% RSLogix 500 project I2P JOB 15 - SOLUTION.RSS, saved by version 10.00.00.00 %
PROJECT "UNTITLED"    % processor: Bul.1763 MicroLogix 1100 Series B %

PROGRAM FILES
  LAD 2   16 rungs

DATA FILES
  O0 OUTPUT  4 elements
  I1 INPUT  6 elements
  S2 STATUS  66 elements
  B3 BINARY  1 elements
  T4 TIMER  1 elements
  C5 COUNTER  1 elements
  R6 CONTROL  1 elements
  N7 INTEGER  1 elements
  F8 FLOAT  1 elements

LADDER 2
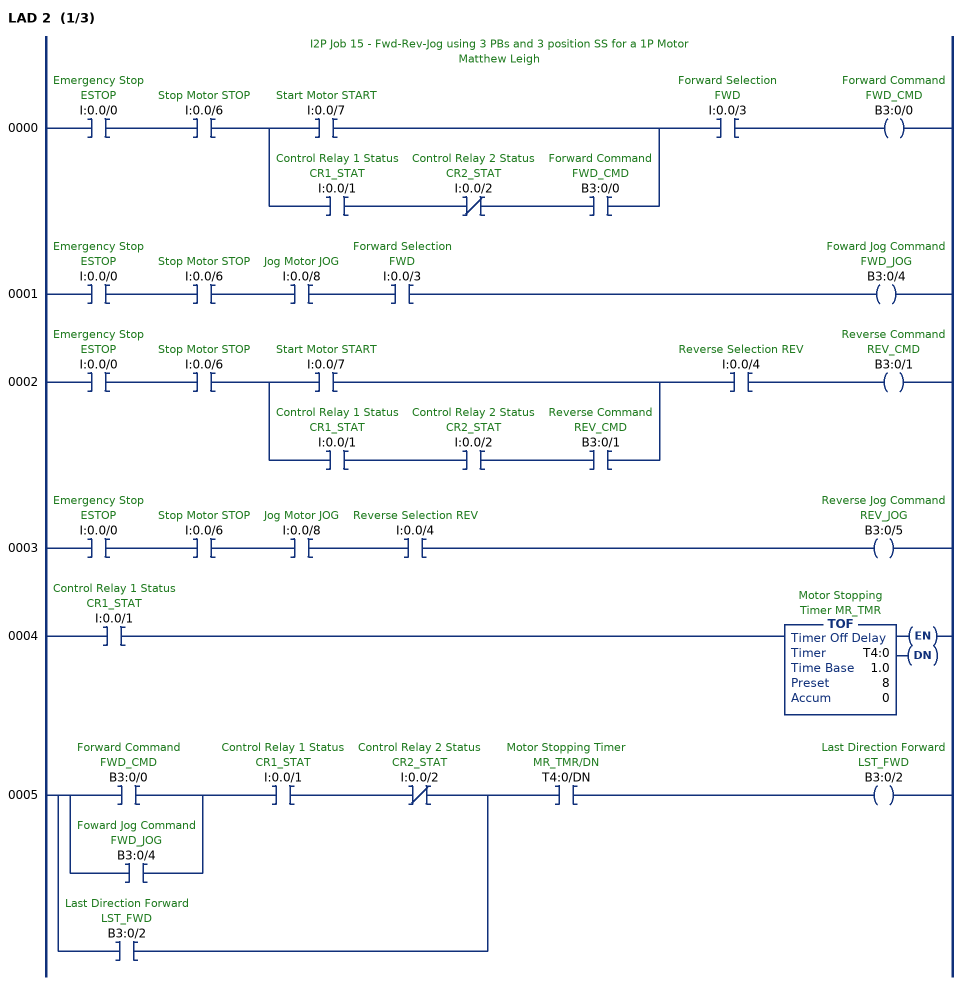
% Rung: 0 %
% I2P Job 15 - Fwd-Rev-Jog using 3 PBs and 3 position SS for a 1P Motor
% Matthew Leigh %
SOR XIC I:0.0/0 XIC I:0.0/6 BST XIC I:0.0/7 NXB XIC I:0.0/1 XIO I:0.0/2 XIC B3:0/0 BND XIC I:0.0/3 OTE B3:0/0 EOR
%   I:0.0/0  ESTOP  "Emergency Stop" %
%   I:0.0/6  STOP  "Stop Motor" %
%   I:0.0/7  START  "Start Motor" %
%   I:0.0/1  CR1_STAT  "Control Relay 1 Status" %
%   I:0.0/2  CR2_STAT  "Control Relay 2 Status" %
%   B3:0/0  FWD_CMD  "Forward Command" %
%   I:0.0/3  FWD  "Forward Selection" %
% Rung: 1 %
SOR XIC I:0.0/0 XIC I:0.0/6 XIC I:0.0/8 XIC I:0.0/3 OTE B3:0/4 EOR
%   I:0.0/0  ESTOP  "Emergency Stop" %
%   I:0.0/6  STOP  "Stop Motor" %
%   I:0.0/8  JOG  "Jog Motor" %
%   I:0.0/3  FWD  "Forward Selection" %
%   B3:0/4  FWD_JOG  "Foward Jog Command" %
% Rung: 2 %
SOR XIC I:0.0/0 XIC I:0.0/6 BST XIC I:0.0/7 NXB XIC I:0.0/1 XIC I:0.0/2 XIC B3:0/1 BND XIC I:0.0/4 OTE B3:0/1 EOR
%   I:0.0/0  ESTOP  "Emergency Stop" %
%   I:0.0/6  STOP  "Stop Motor" %
%   I:0.0/7  START  "Start Motor" %
%   I:0.0/1  CR1_STAT  "Control Relay 1 Status" %
%   I:0.0/2  CR2_STAT  "Control Relay 2 Status" %
%   B3:0/1  REV_CMD  "Reverse Command" %
%   I:0.0/4  REV  "Reverse Selection" %
% Rung: 3 %
SOR XIC I:0.0/0 XIC I:0.0/6 XIC I:0.0/8 XIC I:0.0/4 OTE B3:0/5 EOR
%   I:0.0/0  ESTOP  "Emergency Stop" %
%   I:0.0/6  STOP  "Stop Motor" %
%   I:0.0/8  JOG  "Jog Motor" %
%   I:0.0/4  REV  "Reverse Selection" %
%   B3:0/5  REV_JOG  "Reverse Jog Command" %
% Rung: 4 %
SOR XIC I:0.0/1 TOF T4:0 1.0 8 0 EOR
%   I:0.0/1  CR1_STAT  "Control Relay 1 Status" %
%   T4:0  MR_TMR  "Motor Stopping Timer" %
% Rung: 5 %
SOR BST BST XIC B3:0/0 NXB XIC B3:0/4 BND XIC I:0.0/1 XIO I:0.0/2 NXB XIC B3:0/2 BND XIC T4:0/DN OTE B3:0/2 EOR
%   B3:0/0  FWD_CMD  "Forward Command" %
%   B3:0/4  FWD_JOG  "Foward Jog Command" %
%   I:0.0/1  CR1_STAT  "Control Relay 1 Status" %
%   I:0.0/2  CR2_STAT  "Control Relay 2 Status" %
%   B3:0/2  LST_FWD  "Last Direction Forward" %
%   T4:0  MR_TMR  "Motor Stopping Timer" %

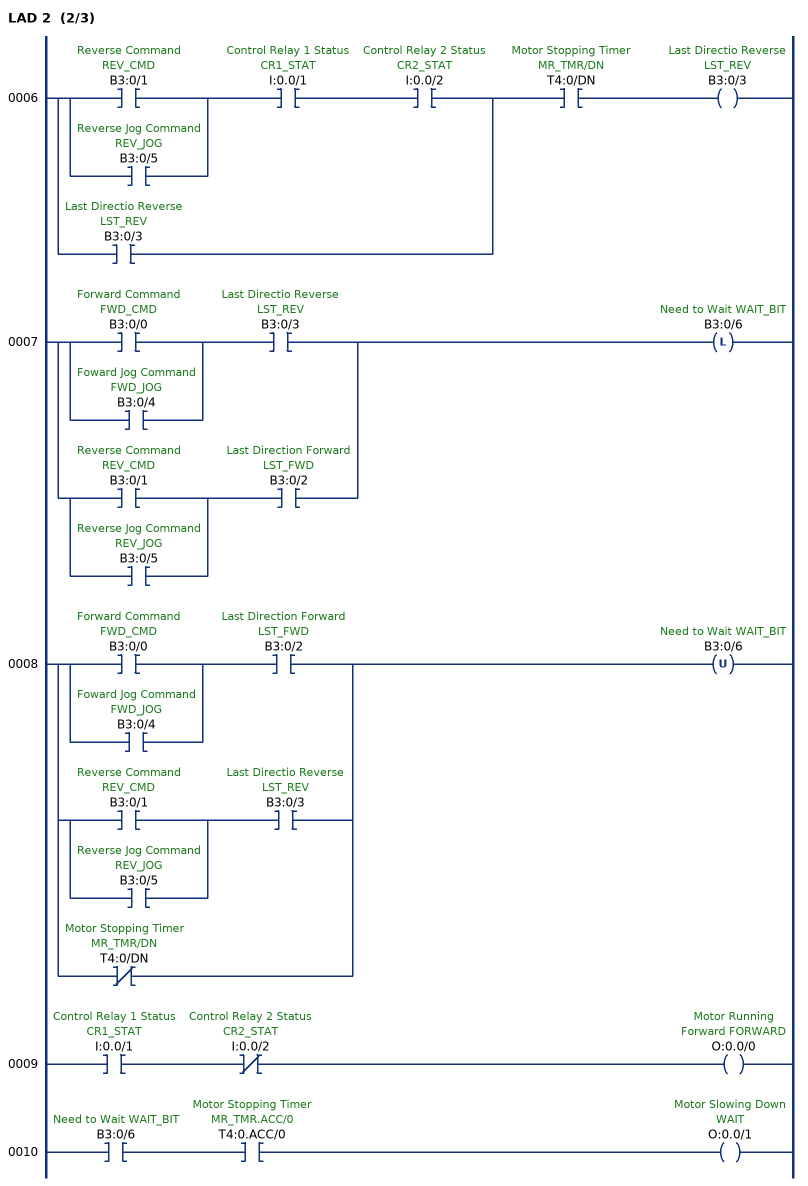
% Rung: 6 %
SOR BST BST XIC B3:0/1 NXB XIC B3:0/5 BND XIC I:0.0/1 XIC I:0.0/2 NXB XIC B3:0/3 BND XIC T4:0/DN OTE B3:0/3 EOR
%   B3:0/1  REV_CMD  "Reverse Command" %
%   B3:0/5  REV_JOG  "Reverse Jog Command" %
%   I:0.0/1  CR1_STAT  "Control Relay 1 Status" %
%   I:0.0/2  CR2_STAT  "Control Relay 2 Status" %
%   B3:0/3  LST_REV  "Last Directio Reverse" %
%   T4:0  MR_TMR  "Motor Stopping Timer" %
% Rung: 7 %
SOR BST BST XIC B3:0/0 NXB XIC B3:0/4 BND XIC B3:0/3 NXB BST XIC B3:0/1 NXB XIC B3:0/5 BND XIC B3:0/2 BND OTL B3:0/6 EOR
%   B3:0/0  FWD_CMD  "Forward Command" %
%   B3:0/4  FWD_JOG  "Foward Jog Command" %
%   B3:0/3  LST_REV  "Last Directio Reverse" %
%   B3:0/1  REV_CMD  "Reverse Command" %
%   B3:0/5  REV_JOG  "Reverse Jog Command" %
%   B3:0/2  LST_FWD  "Last Direction Forward" %
%   B3:0/6  WAIT_BIT  "Need to Wait" %
% Rung: 8 %
SOR BST BST XIC B3:0/0 NXB XIC B3:0/4 BND XIC B3:0/2 NXB BST XIC B3:0/1 NXB XIC B3:0/5 BND XIC B3:0/3 NXB XIO T4:0/DN BND OTU B3:0/6 EOR
%   B3:0/0  FWD_CMD  "Forward Command" %
%   B3:0/4  FWD_JOG  "Foward Jog Command" %
%   B3:0/2  LST_FWD  "Last Direction Forward" %
%   B3:0/1  REV_CMD  "Reverse Command" %
%   B3:0/5  REV_JOG  "Reverse Jog Command" %
%   B3:0/3  LST_REV  "Last Directio Reverse" %
%   T4:0  MR_TMR  "Motor Stopping Timer" %
%   B3:0/6  WAIT_BIT  "Need to Wait" %
% Rung: 9 %
SOR XIC I:0.0/1 XIO I:0.0/2 OTE O:0.0/0 EOR
%   I:0.0/1  CR1_STAT  "Control Relay 1 Status" %
%   I:0.0/2  CR2_STAT  "Control Relay 2 Status" %
%   O:0.0/0  FORWARD  "Motor Running Forward" %
% Rung: 10 %
SOR XIC B3:0/6 XIC T4:0.ACC/0 OTE O:0.0/1 EOR
%   B3:0/6  WAIT_BIT  "Need to Wait" %
%   T4:0  MR_TMR  "Motor Stopping Timer" %
%   O:0.0/1  WAIT  "Motor Slowing Down" %

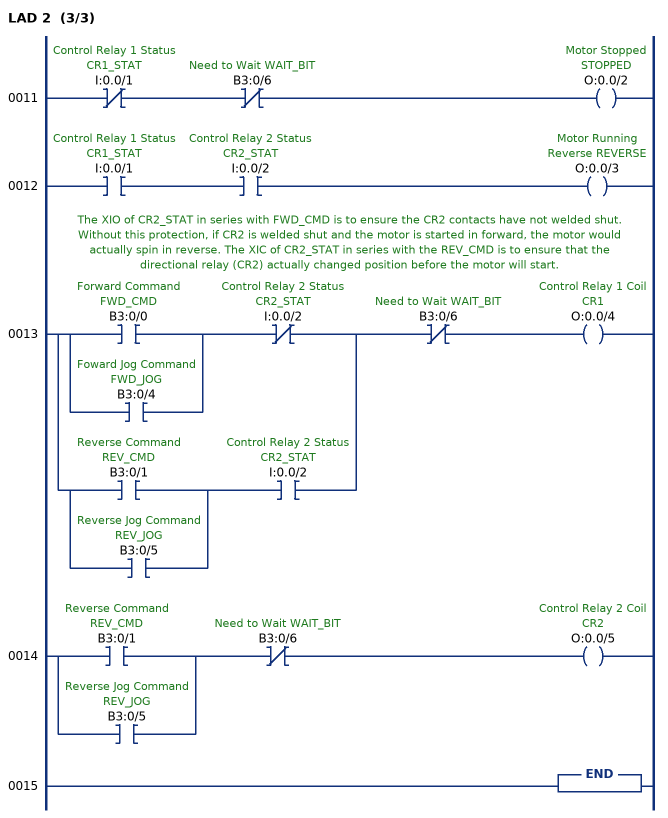
% Rung: 11 %
SOR XIO I:0.0/1 XIO B3:0/6 OTE O:0.0/2 EOR
%   I:0.0/1  CR1_STAT  "Control Relay 1 Status" %
%   B3:0/6  WAIT_BIT  "Need to Wait" %
%   O:0.0/2  STOPPED  "Motor Stopped" %
% Rung: 12 %
SOR XIC I:0.0/1 XIC I:0.0/2 OTE O:0.0/3 EOR
%   I:0.0/1  CR1_STAT  "Control Relay 1 Status" %
%   I:0.0/2  CR2_STAT  "Control Relay 2 Status" %
%   O:0.0/3  REVERSE  "Motor Running Reverse" %
% Rung: 13 %
% The XIO of CR2_STAT in series with FWD_CMD is to ensure the CR2 contacts have not welded shut. Without this protection, if CR2 is welded shut and the motor is started in forward, the motor would actually spin in reverse. The XIC of CR2_STAT in series with the REV_CMD is to ensure that the directional relay (CR2) actually changed position before the motor will start. %
SOR BST BST XIC B3:0/0 NXB XIC B3:0/4 BND XIO I:0.0/2 NXB BST XIC B3:0/1 NXB XIC B3:0/5 BND XIC I:0.0/2 BND XIO B3:0/6 OTE O:0.0/4 EOR
%   B3:0/0  FWD_CMD  "Forward Command" %
%   B3:0/4  FWD_JOG  "Foward Jog Command" %
%   I:0.0/2  CR2_STAT  "Control Relay 2 Status" %
%   B3:0/1  REV_CMD  "Reverse Command" %
%   B3:0/5  REV_JOG  "Reverse Jog Command" %
%   B3:0/6  WAIT_BIT  "Need to Wait" %
%   O:0.0/4  CR1  "Control Relay 1 Coil" %
% Rung: 14 %
SOR BST XIC B3:0/1 NXB XIC B3:0/5 BND XIO B3:0/6 OTE O:0.0/5 EOR
%   B3:0/1  REV_CMD  "Reverse Command" %
%   B3:0/5  REV_JOG  "Reverse Jog Command" %
%   B3:0/6  WAIT_BIT  "Need to Wait" %
%   O:0.0/5  CR2  "Control Relay 2 Coil" %
% Rung: 15 %
SOR END EOR

OTHER DOCUMENTED ADDRESSES
  I:0.0/5  MODE  "Run/Jog Selector A=Run(1) & B=Jog(0)"

DATA TABLE (non-zero values as saved)
DATA T4
% .PRE .ACC %
% T4:0 % 8 0
